# B&R Automation Studio project DosatorePdS
Automation Studio 4.9.6.42 SP; technology packages: mapp 5.24.2, mappView 5.24.0

## Configuration Config1

CPU X20CP1301, AutomationRuntime E4.83, Build 4.1.2, Vc V4.72.6

### Task classes (Cpu.sw)
```
Cyclic#1:
  Program <- Program.prg
Cyclic#4:
  Recipe <- Recipe.prg
Binaries: FWRules, mvLoader, udbdef, TCData, arsvcreg, iomap, sysconf, asfw, User, arconfig, ashwd, Role, ashwac, asnxdb1, Config
Libraries: standard, MpRecipe, MpBase, sys_lib, runtime, MpFile, FileIO, asieccon, astime, arssl, asusb, asbrstr
```

### Hardware
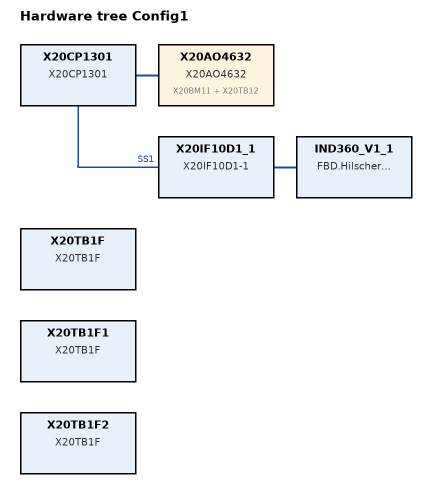
```
IND360_V1_1 : FBD.Hilscher.EIGenEDSAdapterDTM.IND360 V1.1 v1.1 (OrderNumber=IND360 V1.1, VendorAddress=192.168.10.2)  [EIP1 -> X20IF10D1_1.IF1]
  DtmId = a24ae709-e73d-4013-bb43-1e95cdfb2512
  ChannelBlocks_b1ae809b-d69f-462c-9f47-1551c55d3122  // Module 0
  IO_InputImage_b1ae809b-d69f-462c-9f47-1551c55d3122  // 16 Byte(s)
  Channel_1_IO_InputImage_b1ae809b-d69f-462c-9f47-1551c55d3122
  Name_Channel_1_IO_InputImage_b1ae809b-d69f-462c-9f47-1551c55d3122 = MB1_Command_Value
  Type_Channel_1_IO_InputImage_b1ae809b-d69f-462c-9f47-1551c55d3122 = REAL
  Channel_2_IO_InputImage_b1ae809b-d69f-462c-9f47-1551c55d3122
  Name_Channel_2_IO_InputImage_b1ae809b-d69f-462c-9f47-1551c55d3122 = MB1_Channel_Mask
  Type_Channel_2_IO_InputImage_b1ae809b-d69f-462c-9f47-1551c55d3122 = UINT
  Channel_3_IO_InputImage_b1ae809b-d69f-462c-9f47-1551c55d3122
  Name_Channel_3_IO_InputImage_b1ae809b-d69f-462c-9f47-1551c55d3122 = MB1_Command
  Type_Channel_3_IO_InputImage_b1ae809b-d69f-462c-9f47-1551c55d3122 = INT
  Channel_4_IO_InputImage_b1ae809b-d69f-462c-9f47-1551c55d3122
  Name_Channel_4_IO_InputImage_b1ae809b-d69f-462c-9f47-1551c55d3122 = SB1_Reserved_1
  Type_Channel_4_IO_InputImage_b1ae809b-d69f-462c-9f47-1551c55d3122 = INT
  Channel_5_IO_InputImage_b1ae809b-d69f-462c-9f47-1551c55d3122
  Name_Channel_5_IO_InputImage_b1ae809b-d69f-462c-9f47-1551c55d3122 = SB1_Reserved_2
  Type_Channel_5_IO_InputImage_b1ae809b-d69f-462c-9f47-1551c55d3122 = INT
  Channel_6_IO_InputImage_b1ae809b-d69f-462c-9f47-1551c55d3122
  Name_Channel_6_IO_InputImage_b1ae809b-d69f-462c-9f47-1551c55d3122 = SB1_Reserved_3
  Type_Channel_6_IO_InputImage_b1ae809b-d69f-462c-9f47-1551c55d3122 = INT
  Channel_7_IO_InputImage_b1ae809b-d69f-462c-9f47-1551c55d3122
  Name_Channel_7_IO_InputImage_b1ae809b-d69f-462c-9f47-1551c55d3122 = SB1_Command
  Type_Channel_7_IO_InputImage_b1ae809b-d69f-462c-9f47-1551c55d3122 = INT
  IO_OutputImage_b1ae809b-d69f-462c-9f47-1551c55d3122  // 16 Byte(s)
  Channel_1_IO_OutputImage_b1ae809b-d69f-462c-9f47-1551c55d3122
  Name_Channel_1_IO_OutputImage_b1ae809b-d69f-462c-9f47-1551c55d3122 = MB1_Measuring_Value
  Type_Channel_1_IO_OutputImage_b1ae809b-d69f-462c-9f47-1551c55d3122 = REAL
  Channel_2_IO_OutputImage_b1ae809b-d69f-462c-9f47-1551c55d3122
  Name_Channel_2_IO_OutputImage_b1ae809b-d69f-462c-9f47-1551c55d3122 = MB1_Device_Status
  Type_Channel_2_IO_OutputImage_b1ae809b-d69f-462c-9f47-1551c55d3122 = UINT
  Channel_3_IO_OutputImage_b1ae809b-d69f-462c-9f47-1551c55d3122
  Name_Channel_3_IO_OutputImage_b1ae809b-d69f-462c-9f47-1551c55d3122 = MB1_Response
  Type_Channel_3_IO_OutputImage_b1ae809b-d69f-462c-9f47-1551c55d3122 = INT
  Channel_4_IO_OutputImage_b1ae809b-d69f-462c-9f47-1551c55d3122
  Name_Channel_4_IO_OutputImage_b1ae809b-d69f-462c-9f47-1551c55d3122 = SB1_Status_Group_1
  Type_Channel_4_IO_OutputImage_b1ae809b-d69f-462c-9f47-1551c55d3122 = INT
  Channel_5_IO_OutputImage_b1ae809b-d69f-462c-9f47-1551c55d3122
  Name_Channel_5_IO_OutputImage_b1ae809b-d69f-462c-9f47-1551c55d3122 = SB1_Status_Group_2
  Type_Channel_5_IO_OutputImage_b1ae809b-d69f-462c-9f47-1551c55d3122 = INT
  Channel_6_IO_OutputImage_b1ae809b-d69f-462c-9f47-1551c55d3122
  Name_Channel_6_IO_OutputImage_b1ae809b-d69f-462c-9f47-1551c55d3122 = SB1_Status_Group_3
  Type_Channel_6_IO_OutputImage_b1ae809b-d69f-462c-9f47-1551c55d3122 = INT
  Channel_7_IO_OutputImage_b1ae809b-d69f-462c-9f47-1551c55d3122
  Name_Channel_7_IO_OutputImage_b1ae809b-d69f-462c-9f47-1551c55d3122 = SB1_Response
  Type_Channel_7_IO_OutputImage_b1ae809b-d69f-462c-9f47-1551c55d3122 = INT
X20AO4632 : X20AO4632 v1.3.1.0  [SS1 -> X20TB12.SS; SL -> X20BM11.SL1]
  ChannelType01 = 0 to 20mA
X20BM11 : X20BM11 v1.1.0.0  [X2X1 -> X20CP1301.IF6]
X20CP1301 : X20CP1301 v1.7.0.0  [X1 -> X1.SL; X2 -> X2.SL; X3 -> X3.SL]
  Module X1 (Type=X1, Virtual=true, Version=1.7.0.0)
    Connection (Connector=SS1, TargetModule=X20TB1F, TargetConnector=SS)
    Connection (Connector=SL, TargetModule=X20CP1301, TargetConnector=X1)
    X1AI_ChannelType01 = 0 to 20mA
    X1AI1_InputFilter = level 2
    X1AI_ChannelType02 = 0 to 20mA
  Module X2 (Type=X2, Virtual=true, Version=1.7.0.0)
    Connection (Connector=SS1, TargetModule=X20TB1F1, TargetConnector=SS)
    Connection (Connector=SL, TargetModule=X20CP1301, TargetConnector=X2)
  Module X3 (Type=X3, Virtual=true, Version=1.7.0.0)
    Connection (Connector=SS1, TargetModule=X20TB1F2, TargetConnector=SS)
    Connection (Connector=SL, TargetModule=X20CP1301, TargetConnector=X3)
  Connector IF2:
    ActivateDevice = 1
    Mode = Manual
    InternetAddress = 192.168.0.2
    SubnetMask = 255.255.255.0
  ConfigurationID = DosatorePdS_Config1
  UserPartitionSize = 200
  EnableUsbRemoteInstall = 1
  Cyclic1Tolerance = 0
  FileDevice1
  FileDeviceName1 = CF
  FileDevicePath1 = F:\Recipe
  FtpUser1
  FtpUsername1 = bazzica
  FtpUserPassword1 = htUSodyHi80qCEfYHuTU7vQ0j0QXP3jVAlZaBuEyoRs=  // promass
  FtpUserSalt1 = 1uLtMhRf
  FTPAccessRight1 = 0
  ActivateOpcUa = 1
  OpcUaInformationModels_PV_Version = 1
X20IF10D1_1 : X20IF10D1-1 v1.7.0.0  [SS -> X20CP1301.SS1]
  Connector IF1:
    DtmId = ce78e8b2-5855-467c-9c90-e15d78aa6884
  ConfigFile = X20IF10D1_1.dtm
  ConfigModule = asnxdb1
X20TB12 : X20TB12 v1.0.0.0
X20TB1F : X20TB1F v1.0.0.0
X20TB1F1 : X20TB1F v1.0.0.0
X20TB1F2 : X20TB1F v1.0.0.0
```

### IoMap.iom - X20CP1301/IoMap.iom
```iecst
VAR_CONFIG
	Cyclic#1.GlbIO.Ao.Valvola AT %QW."X20AO4632".AnalogOutput01;
	GlbIO.Do.PompaAspirazione AT %QX."X3".DigitalOutput01;
	PesoBilancia_G AT %ID."IND360_V1_1".MB1_Command_Value;
	::GlbIO.Ai.Valvola AT %IW."X1".AnalogInput02;
END_VAR
```

## Configuration Config2

### Task classes (Cpu.sw)
```
Cyclic#1:
  simu <- simu.prg
  Program <- Program.prg
Cyclic#4:
  Recipe <- Recipe.prg
Binaries: FWRules, mvLoader, udbdef, TCData, arsvcreg, iomap, sysconf, asfw, User, arconfig, ashwd, Role, ashwac, asnxdb1, Config
Libraries: standard, MpRecipe, MpBase, sys_lib, runtime, MpFile, FileIO, asieccon, astime, arssl, asusb, asbrstr
```

### Hardware
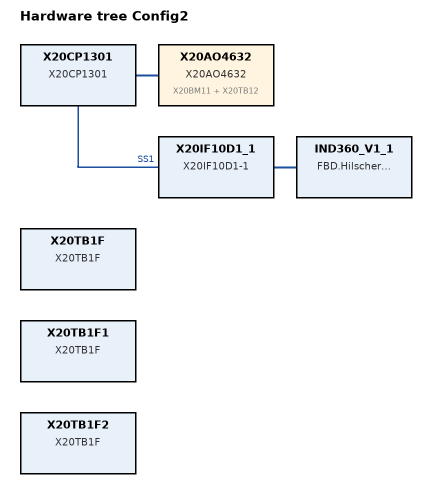
```
IND360_V1_1 : FBD.Hilscher.EIGenEDSAdapterDTM.IND360 V1.1 v1.1 (OrderNumber=IND360 V1.1, VendorAddress=192.168.10.2)  [EIP1 -> X20IF10D1_1.IF1]
  DtmId = a24ae709-e73d-4013-bb43-1e95cdfb2512
  ChannelBlocks_b1ae809b-d69f-462c-9f47-1551c55d3122  // Module 0
  IO_InputImage_b1ae809b-d69f-462c-9f47-1551c55d3122  // 16 Byte(s)
  Channel_1_IO_InputImage_b1ae809b-d69f-462c-9f47-1551c55d3122
  Name_Channel_1_IO_InputImage_b1ae809b-d69f-462c-9f47-1551c55d3122 = MB1_Command_Value
  Type_Channel_1_IO_InputImage_b1ae809b-d69f-462c-9f47-1551c55d3122 = REAL
  Channel_2_IO_InputImage_b1ae809b-d69f-462c-9f47-1551c55d3122
  Name_Channel_2_IO_InputImage_b1ae809b-d69f-462c-9f47-1551c55d3122 = MB1_Channel_Mask
  Type_Channel_2_IO_InputImage_b1ae809b-d69f-462c-9f47-1551c55d3122 = UINT
  Channel_3_IO_InputImage_b1ae809b-d69f-462c-9f47-1551c55d3122
  Name_Channel_3_IO_InputImage_b1ae809b-d69f-462c-9f47-1551c55d3122 = MB1_Command
  Type_Channel_3_IO_InputImage_b1ae809b-d69f-462c-9f47-1551c55d3122 = INT
  Channel_4_IO_InputImage_b1ae809b-d69f-462c-9f47-1551c55d3122
  Name_Channel_4_IO_InputImage_b1ae809b-d69f-462c-9f47-1551c55d3122 = SB1_Reserved_1
  Type_Channel_4_IO_InputImage_b1ae809b-d69f-462c-9f47-1551c55d3122 = INT
  Channel_5_IO_InputImage_b1ae809b-d69f-462c-9f47-1551c55d3122
  Name_Channel_5_IO_InputImage_b1ae809b-d69f-462c-9f47-1551c55d3122 = SB1_Reserved_2
  Type_Channel_5_IO_InputImage_b1ae809b-d69f-462c-9f47-1551c55d3122 = INT
  Channel_6_IO_InputImage_b1ae809b-d69f-462c-9f47-1551c55d3122
  Name_Channel_6_IO_InputImage_b1ae809b-d69f-462c-9f47-1551c55d3122 = SB1_Reserved_3
  Type_Channel_6_IO_InputImage_b1ae809b-d69f-462c-9f47-1551c55d3122 = INT
  Channel_7_IO_InputImage_b1ae809b-d69f-462c-9f47-1551c55d3122
  Name_Channel_7_IO_InputImage_b1ae809b-d69f-462c-9f47-1551c55d3122 = SB1_Command
  Type_Channel_7_IO_InputImage_b1ae809b-d69f-462c-9f47-1551c55d3122 = INT
  IO_OutputImage_b1ae809b-d69f-462c-9f47-1551c55d3122  // 16 Byte(s)
  Channel_1_IO_OutputImage_b1ae809b-d69f-462c-9f47-1551c55d3122
  Name_Channel_1_IO_OutputImage_b1ae809b-d69f-462c-9f47-1551c55d3122 = MB1_Measuring_Value
  Type_Channel_1_IO_OutputImage_b1ae809b-d69f-462c-9f47-1551c55d3122 = REAL
  Channel_2_IO_OutputImage_b1ae809b-d69f-462c-9f47-1551c55d3122
  Name_Channel_2_IO_OutputImage_b1ae809b-d69f-462c-9f47-1551c55d3122 = MB1_Device_Status
  Type_Channel_2_IO_OutputImage_b1ae809b-d69f-462c-9f47-1551c55d3122 = UINT
  Channel_3_IO_OutputImage_b1ae809b-d69f-462c-9f47-1551c55d3122
  Name_Channel_3_IO_OutputImage_b1ae809b-d69f-462c-9f47-1551c55d3122 = MB1_Response
  Type_Channel_3_IO_OutputImage_b1ae809b-d69f-462c-9f47-1551c55d3122 = INT
  Channel_4_IO_OutputImage_b1ae809b-d69f-462c-9f47-1551c55d3122
  Name_Channel_4_IO_OutputImage_b1ae809b-d69f-462c-9f47-1551c55d3122 = SB1_Status_Group_1
  Type_Channel_4_IO_OutputImage_b1ae809b-d69f-462c-9f47-1551c55d3122 = INT
  Channel_5_IO_OutputImage_b1ae809b-d69f-462c-9f47-1551c55d3122
  Name_Channel_5_IO_OutputImage_b1ae809b-d69f-462c-9f47-1551c55d3122 = SB1_Status_Group_2
  Type_Channel_5_IO_OutputImage_b1ae809b-d69f-462c-9f47-1551c55d3122 = INT
  Channel_6_IO_OutputImage_b1ae809b-d69f-462c-9f47-1551c55d3122
  Name_Channel_6_IO_OutputImage_b1ae809b-d69f-462c-9f47-1551c55d3122 = SB1_Status_Group_3
  Type_Channel_6_IO_OutputImage_b1ae809b-d69f-462c-9f47-1551c55d3122 = INT
  Channel_7_IO_OutputImage_b1ae809b-d69f-462c-9f47-1551c55d3122
  Name_Channel_7_IO_OutputImage_b1ae809b-d69f-462c-9f47-1551c55d3122 = SB1_Response
  Type_Channel_7_IO_OutputImage_b1ae809b-d69f-462c-9f47-1551c55d3122 = INT
X20AO4632 : X20AO4632 v1.3.1.0  [SS1 -> X20TB12.SS; SL -> X20BM11.SL1]
  ChannelType01 = 0 to 20mA
X20BM11 : X20BM11 v1.1.0.0  [X2X1 -> X20CP1301.IF6]
X20CP1301 : X20CP1301 v1.7.0.0  [X1 -> X1.SL; X2 -> X2.SL; X3 -> X3.SL]
  Module X1 (Type=X1, Virtual=true, Version=1.7.0.0)
    Connection (Connector=SS1, TargetModule=X20TB1F, TargetConnector=SS)
    Connection (Connector=SL, TargetModule=X20CP1301, TargetConnector=X1)
    X1AI_ChannelType01 = 0 to 20mA
    X1AI1_InputFilter = level 2
    X1AI_ChannelType02 = 0 to 20mA
  Module X2 (Type=X2, Virtual=true, Version=1.7.0.0)
    Connection (Connector=SS1, TargetModule=X20TB1F1, TargetConnector=SS)
    Connection (Connector=SL, TargetModule=X20CP1301, TargetConnector=X2)
  Module X3 (Type=X3, Virtual=true, Version=1.7.0.0)
    Connection (Connector=SS1, TargetModule=X20TB1F2, TargetConnector=SS)
    Connection (Connector=SL, TargetModule=X20CP1301, TargetConnector=X3)
  Connector IF2:
    ActivateDevice = 1
    Mode = Manual
    InternetAddress = 192.168.0.2
    SubnetMask = 255.255.255.0
  ConfigurationID = DosatorePdS_Config1
  UserPartitionSize = 200
  Simulation = 1
  EnableUsbRemoteInstall = 1
  Cyclic1Tolerance = 0
  FileDevice1
  FileDeviceName1 = CF
  FileDevicePath1 = F:\Recipe
  FtpUser1
  FtpUsername1 = bazzica
  FtpUserPassword1 = htUSodyHi80qCEfYHuTU7vQ0j0QXP3jVAlZaBuEyoRs=  // promass
  FtpUserSalt1 = 1uLtMhRf
  FTPAccessRight1 = 0
  ActivateOpcUa = 1
  OpcUaInformationModels_PV_Version = 1
X20IF10D1_1 : X20IF10D1-1 v1.7.0.0  [SS -> X20CP1301.SS1]
  Connector IF1:
    DtmId = ce78e8b2-5855-467c-9c90-e15d78aa6884
  ConfigFile = X20IF10D1_1.dtm
  ConfigModule = asnxdb1
X20TB12 : X20TB12 v1.0.0.0
X20TB1F : X20TB1F v1.0.0.0
X20TB1F1 : X20TB1F v1.0.0.0
X20TB1F2 : X20TB1F v1.0.0.0
```

### IoMap.iom - X20CP1301/IoMap.iom
```iecst
VAR_CONFIG
	Cyclic#1.GlbIO.Ao.Valvola AT %QW."X20AO4632".AnalogOutput01;
	GlbIO.Do.PompaAspirazione AT %QX."X3".DigitalOutput01;
END_VAR
```

## Logical view

Binary libraries used (declarations not repeated): operator, runtime, astime, AsIecCon, standard, MpRecipe 5.24.2, MpBase 5.24.1, sys_lib, MpFile 5.24.2, FileIO

### Global.typ - Global data types
```iecst
TYPE
	TypDo : 	STRUCT
		PompaAspirazione : BOOL;
	END_STRUCT;
	TypAi : 	STRUCT
		Valvola : INT;
		Bilancia : INT;
	END_STRUCT;
	TypAo : 	STRUCT
		Valvola : INT;
	END_STRUCT;
	TypIO : 	STRUCT
		Ai : TypAi;
		Ao : TypAo;
		Do : TypDo;
	END_STRUCT;
	Typ_recipe : 	STRUCT
		PesoRichiesto : REAL;
		fPesoAnticipoChiusura : REAL;
		fSogliaDosaggioLento : REAL;
		fSogliaMicrodosaggio : REAL;
		fPercentualeValvolaVeloce : REAL;
		fPercentualeValvolaLenta : REAL;
		fPercentualeValvolaFine : REAL;
		fFattoreCorrezione : REAL;
	END_STRUCT;
END_TYPE
```

### Global.var - Global variables
```iecst
VAR
	GlbIO : TypIO;
	Recipe : Typ_recipe;
	PesoBilancia_G : REAL; (*// Peso finale in grammi*)
END_VAR
```


### Program Logical/Program (IEC)

#### Cyclic.st - Cyclic code
```iecst
PROGRAM _CYCLIC
// #######################################################################
// --- LOGICA PRINCIPALE E CALIBRAZIONE ---
// #######################################################################

	IF PercentualeValvola > 0 THEN
		radialGauge := REAL_TO_INT(PercentualeValvola*10);
	ELSE
		radialGauge := 0;
	END_IF

	// conversione segnale d'ingresso valvola

	PercentualeValvola := (((INT_TO_REAL(GlbIO.Ai.Valvola) - 6553.0) / (32767.0 - 6553.0)) * 100.0);

// --- ESECUZIONE TIMER ---
	TON_AttesaStabilizzazione(IN := bStartTimerCal, PT := REAL_TO_TIME(fDurataTestSec * 1000.0));
	TON_AttesaStabilizzazione;

	// --- MAPPATURA I/O e CHIAMATA AL BLOCCO FUNZIONE ---
	PesoBilancia_AI := GlbIO.Ai.Bilancia;
	GlbIO.Ao.Valvola := REAL_TO_INT(Valvola_AO);

	IF Pulsante_Tara THEN Pulsante_Tara := FALSE; PesoTara := PesoBilancia_G; END_IF
	PesoBilancia_G := PesoBilancia_G - PesoTara;

	IF Stop_HMI THEN Dosatore.bFermaDosaggo := 1; ELSE Dosatore.bFermaDosaggo := 0; END_IF
	TON_timerDosaggio;
	TON_timerDosaggio.PT := T#500s;

	IF NOT (Dosatore.eStatoDosaggio = eST_ERRORE OR Dosatore.eStatoDosaggio = eST_COMPLETATO OR Dosatore.eStatoDosaggio = eST_IDLE) THEN
		TON_timerDosaggio.IN := TRUE;
		tDosaggio_HMI := TIME_TO_REAL(TON_timerDosaggio.ET) / 1000;
	ELSE
		TON_timerDosaggio.IN := FALSE;
	END_IF

	Dosatore.fPesoAnticipoChiusura 			:= Recipe.fPesoAnticipoChiusura;
	Dosatore.fSogliaDosaggioLento 			:= Recipe.fSogliaDosaggioLento;
	Dosatore.fSogliaMicrodosaggio 			:= Recipe.fSogliaMicrodosaggio;
	Dosatore.fPercentualeValvolaVeloce 		:= Recipe.fPercentualeValvolaVeloce;
	Dosatore.fPercentualeValvolaLenta 		:= Recipe.fPercentualeValvolaLenta;
	Dosatore.fPercentualeValvolaFine 		:= Recipe.fPercentualeValvolaFine;
	Dosatore.fFattoreCorrezione 			:= Recipe.fFattoreCorrezione;
	Dosatore.fFeadbackValvolaProporzionale 	:= PercentualeValvola;
	PesoRichiesto_HMI						:= Recipe.PesoRichiesto;

	Dosatore(
		fPesoAttualeBilancia := PesoBilancia_G,
		fPesoRichiesto := PesoRichiesto_HMI,
		bAvviaDosaggio := StartDosaggio_HMI
		);

	Recipe.fPesoAnticipoChiusura := Dosatore.fPesoAnticipoChiusura;

	BilanciaManager(
		iRawInput := PesoBilancia_AI,
		bComandoTare := Pulsante_Tara
		// fCapacitaMaxG e iRawMax usano i valori di default (5000.0, 32767) se non specificati
		);

	// Mappa l'uscita
	// PesoBilancia_G := BilanciaManager.fPesoGrammi;

	Valvola_AO := (Dosatore.fUscitaValvolaProporzionale * (32767 - 6600) / 100) + 6600;

	// --- SEQUENZA DI MISURAZIONE DELLA PORTATA ---
	// Logica per eseguire il test di portata con Timer e chiusura valvola
	IF eStatoCalibrazione = eCAL_TEST_PUNTO1_BASSO OR eStatoCalibrazione = eCAL_TEST_PUNTO2_ALTO THEN
	(*	bStartTimerCal := FALSE;*)
		IF NOT TON_AttesaStabilizzazione.Q THEN
			// La variabile Veloce qui funge da variabile temporanea per l'apertura in test
			GlbIO.Ao.Valvola := REAL_TO_INT(Dosatore.fPercentualeValvolaVeloce * 32767 / 100);
		ELSE
			GlbIO.Ao.Valvola := REAL_TO_INT(10000.0);
		END_IF

		// Calcolo della portata dopo il timeout + 10s di stabilizzazione
		IF TON_AttesaStabilizzazione.Q AND TON_AttesaStabilizzazione.ET >= REAL_TO_TIME((fDurataTestSec) * 1000.0) THEN
			fPortataMisurata := (PesoBilancia_G - fPesoIniziale) / fDurataTestSec;
			bStartTimerCal := FALSE; // Termina il test
		END_IF
	END_IF

	// #######################################################################
	// --- MACCHINA A STATI DI CALIBRAZIONE ---
	// #######################################################################

	IF bStartCalibrazione AND NOT bCalibrazioneCompletata THEN

		CASE eStatoCalibrazione OF

			eCAL_IDLE:
				bStartTimerCal := FALSE;
				//Bilancia.Tare := TRUE;
				Dosatore.fFattoreCorrezione := 0.0; // Disabilita l'auto-tuning
				eStatoCalibrazione := eCAL_PREPARA_TEST;

			eCAL_PREPARA_TEST:
				fPortataMisurata := 0.0;
				fPesoIniziale := 0.0;
				eStatoCalibrazione := eCAL_TEST_PUNTO1_BASSO;

				fPesoIniziale := PesoBilancia_G;
				bStartTimerCal := TRUE;

			eCAL_TEST_PUNTO1_BASSO:
				// TEST 1: Misura della portata al punto P1 (20% apertura)
				Dosatore.fPercentualeValvolaVeloce := fPercentualeTestBasso;

//					fPesoIniziale := PesoBilancia_G;
//					bStartTimerCal := TRUE;
				IF NOT bStartTimerCal AND (fPortataMisurata > 0.0) THEN
					fPortataTestBasso := fPortataMisurata;
					eStatoCalibrazione := eCAL_TEST_PUNTO2_ALTO;

					fPesoIniziale := PesoBilancia_G;
					fPortataMisurata := 0;
					bStartTimerCal := TRUE;
				END_IF

			eCAL_TEST_PUNTO2_ALTO:
				// TEST 2: Misura della portata al punto P2 (80% apertura)
				Dosatore.fPercentualeValvolaVeloce := fPercentualeTestAlto;

//					fPesoIniziale := PesoBilancia_G;
//					bStartTimerCal := TRUE;
				IF NOT bStartTimerCal AND (fPortataMisurata > 0.0) THEN
					fPortataTestAlto := fPortataMisurata;
					eStatoCalibrazione := eCAL_CALCOLA_CURVA;
				END_IF

			eCAL_CALCOLA_CURVA:
				// Calcolo dei coefficienti della curva lineare (Percentuale = m * Portata + q)
				IF (fPortataTestAlto - fPortataTestBasso) > 0.001 THEN
					fPendenza_m := (fPercentualeTestAlto - fPercentualeTestBasso) /
					(fPortataTestAlto - fPortataTestBasso);
					fIntercetta_q := fPercentualeTestBasso - (fPendenza_m * fPortataTestBasso);

					eStatoCalibrazione := eCAL_MISURA_VOLO;
				ELSE
					eStatoCalibrazione := eCAL_ERRORE; // Errore: Le portate sono uguali o zero
				END_IF

			eCAL_MISURA_VOLO:
				// CRUCIALE: Misura il peso in volo (forza Dosatore.fPesoAnticipoChiusura = 0.0)
				Dosatore.fPesoAnticipoChiusura := 0.0;
				fSetPointTaratura := 2000.0;
				PesoRichiesto_HMI := fSetPointTaratura;

				StartDosaggio_HMI := TRUE;

				IF Dosatore.bDosaggioCompletato THEN
					StartDosaggio_HMI := FALSE;
					bStartTimerCal := TRUE;
					eStatoCalibrazione := eCAL_ATTESA_PESO;
				END_IF

			eCAL_ATTESA_PESO:
				// Attende stabilizzazione e calcola il volo
				IF TON_AttesaStabilizzazione.Q THEN
					bStartTimerCal := FALSE;

					fAnticipoMisurato := PesoBilancia_G - fSetPointTaratura;

					IF fAnticipoMisurato < 0.5 THEN fAnticipoMisurato := 0.5; END_IF

					eStatoCalibrazione := eCAL_APPLICA_VALORI;
				END_IF

			eCAL_APPLICA_VALORI:
				// Applica i valori tarati al blocco funzione
				Dosatore.fPesoAnticipoChiusura := fAnticipoMisurato;

				// Applica le percentuali dalla curva di calibrazione:
				Dosatore.fPercentualeValvolaVeloce := (fPendenza_m * fPortataTargetVeloce) + fIntercetta_q;
				Dosatore.fPercentualeValvolaLenta := (fPendenza_m * fPortataTargetLenta) + fIntercetta_q;
				Dosatore.fPercentualeValvolaFine := (fPendenza_m * fPortataTargetFine) + fIntercetta_q;

				// Limitazioni di sicurezza
				IF Dosatore.fPercentualeValvolaVeloce > 100.0 THEN Dosatore.fPercentualeValvolaVeloce := 100.0; END_IF
				IF Dosatore.fPercentualeValvolaFine < 0.0 THEN Dosatore.fPercentualeValvolaFine := 0.0; END_IF

				// Ripristina l'auto-taratura continua
				Dosatore.fFattoreCorrezione := 0.1;

				eStatoCalibrazione := eCAL_COMPLETATO;

			eCAL_COMPLETATO:
				bCalibrazioneCompletata := TRUE;
				eStatoCalibrazione := eCAL_IDLE;

			eCAL_ERRORE:
			// ... Logica di errore

		END_CASE

	END_IF

	IF GlbIO.Ao.Valvola < 6500 THEN GlbIO.Ao.Valvola := 6500; END_IF

END_PROGRAM
```

#### Init.st - Init code
```iecst
PROGRAM _INIT
	(* Insert code here *)

	IF bCalibrazioneCompletata THEN
		// Applica i valori tarati al blocco funzione
		Dosatore.fPesoAnticipoChiusura := fAnticipoMisurato;

		// Applica le percentuali dalla curva di calibrazione:
		Dosatore.fPercentualeValvolaVeloce := (fPendenza_m * fPortataTargetVeloce) + fIntercetta_q;
		Dosatore.fPercentualeValvolaLenta := (fPendenza_m * fPortataTargetLenta) + fIntercetta_q;
		Dosatore.fPercentualeValvolaFine := (fPendenza_m * fPortataTargetFine) + fIntercetta_q;

		// Limitazioni di sicurezza
		IF Dosatore.fPercentualeValvolaVeloce > 100.0 THEN Dosatore.fPercentualeValvolaVeloce := 100.0; END_IF
		IF Dosatore.fPercentualeValvolaFine < 0.0 THEN Dosatore.fPercentualeValvolaFine := 0.0; END_IF

		// Ripristina l'auto-taratura continua
		Dosatore.fFattoreCorrezione := 0.1;
	END_IF

END_PROGRAM
```

#### Types.typ - Local data types
```iecst
TYPE
	enSignalType :
		(
		eST_0_20mA,
		eST_4_20mA
		);
	enStatoDosaggio :
		(
		eST_IDLE := 10,
		eST_VELOCE := 20,
		eST_LENTO := 30,
		eST_FINE := 40,
		eST_ATTESA_STABILIZZAZIONE := 50,
		eST_COMPLETATO := 60,
		eST_ERRORE := 0
		);
	enStatoCalibrazione :
		( (*// Macchina a Stati per la Calibrazione*)
		eCAL_IDLE := 10,
		eCAL_PREPARA_TEST := 20,
		eCAL_TEST_PUNTO1_BASSO,
		eCAL_TEST_PUNTO2_ALTO,
		eCAL_CALCOLA_CURVA,
		eCAL_MISURA_VOLO := 30,
		eCAL_ATTESA_PESO := 40,
		eCAL_APPLICA_VALORI := 50,
		eCAL_COMPLETATO := 60,
		eCAL_ERRORE := 0
		);
END_TYPE
```

#### Variables.var - Local variables
```iecst
VAR
	tDosaggio_HMI : REAL;
	TON_timerDosaggio : TON;
	PercentualeValvola : REAL;
END_VAR
VAR RETAIN
	Dosatore : FB_DosaggioPolvere; (*// Istanza del blocco funzione*)
END_VAR
VAR
	PesoBilancia_AI : INT; (*// Ingresso Analogico (da I/O Link o bus)*)
	Valvola_AO : REAL; (*// Uscita Analogica (verso I/O Link o bus)*)
	Stop_HMI : BOOL;
END_VAR
VAR RETAIN
	PesoRichiesto_HMI : REAL; (*// Setpoint (da HMI)*)
END_VAR
VAR
	StartDosaggio_HMI : BOOL; (*// Tasto Start (da HMI)*)
	DosaggioOK : BOOL; (*// Stato di completamento*) (*// --- VARIABILI PER LA TARATURA AUTOMATICA ---*)
	bStartCalibrazione : BOOL; (*// Comando esterno per avviare la taratura (es. da HMI)*)
END_VAR
VAR RETAIN
	bCalibrazioneCompletata : BOOL;
END_VAR
VAR
	eStatoCalibrazione : enStatoCalibrazione; (*// Macchina a Stati per la Calibrazione*) (*// Variabili interne per la Taratura*)
END_VAR
(*// Parametri della Curva e Portate Target*)
VAR
	fPortataTestBasso : REAL;
	fPortataTestAlto : REAL;
	fPercentualeTestBasso : REAL := 45;
	fPercentualeTestAlto : REAL := 80.0;
END_VAR
VAR RETAIN
	fPendenza_m : REAL;
	fIntercetta_q : REAL;
END_VAR
VAR
	fPortataTargetVeloce : REAL := 80.0; (*// Target di flusso in g/s per Veloce*)
	fPortataTargetLenta : REAL := 15.0; (*// Target di flusso in g/s per Lenta*)
	fPortataTargetFine : REAL := 5.0; (*// Target di flusso in g/s per Fine*)
END_VAR
(*// Variabili interne*)
VAR
	fAnticipoMisurato : REAL; (*// Risultato del test di misurazione del volo*)
	fSetPointTaratura : REAL; (*// Setpoint specifico per il test*)
	fPortataMisurata : REAL; (*// Portata misurata in [grammi/secondo]*)
	fPesoIniziale : REAL;
	fDurataTestSec : REAL := 5; (*// Durata di ogni test di portata (3 secondi)*)
END_VAR
(*// Timer e Logica Timer*)
VAR
	TON_AttesaStabilizzazione : TON; (*// Timer per attendere che la bilancia si stabilizzi*)
	bStartTimerCal : BOOL := FALSE;
	ModuloBilancia_Raw : INT; (*// Dati grezzi in ingresso (dall'I/O)*)
END_VAR
VAR RETAIN
	PesoTara : REAL;
END_VAR
VAR
	Pulsante_Tara : BOOL; (*// Comando di azzeramento da HMI o logica*)
END_VAR
VAR RETAIN
	BilanciaManager : FB_GestioneBilancia; (*// Istanza del Blocco Funzione*)
END_VAR
VAR
	radialGauge : UINT;
END_VAR
```

#### LocalFunctions.fun
```iecst
FUNCTION_BLOCK FB_GestioneBilancia
	VAR_INPUT
		iRawInput : INT; (*// Ingresso: Valore raw (grezzo) letto dal modulo I/O (es. 0 a 32767)*)
		bComandoTare : BOOL; (*// Ingresso: Commuta a TRUE per eseguire l'azzeramento (Tara)*)
		eTipoSegnale : enSignalType := eST_4_20mA; (*/ NUOVO: Tipo di segnale (0-20mA o 4-20mA)*)
		fCapacitaMaxG : REAL := 6000.0; (*// Ingresso: Capacità massima della bilancia in grammi*)
		iRawMax : INT := 32767; (*// Ingresso: Valore massimo raw del modulo I/O*)
	END_VAR
	VAR_OUTPUT
		bErroreSegnale : BOOL;
		fPesoGrammi : REAL; (*// Uscita: Peso convertito e tarato in grammi (REAL)*)
	END_VAR
	VAR
		fFattoreConversione : REAL; (*// Fattore per convertire Raw in Grammi/Volt*)
		fOffsetTara : REAL := 0.0; (*// Offset di tara (peso memorizzato durante l'azzeramento)*)
		fPesoLordoSenzaOffset : REAL; (*// Peso convertito prima dell'applicazione della tara*)
		iRawMin : INT; (*// Valore raw minimo corrispondente a 0mA o 4mA*)
		iRawRange : INT; (*// RawMax - RawMin*)
		fRawAttualeNormalizzato : REAL; (*// Raw letto - RawMin*)
	END_VAR
END_FUNCTION_BLOCK

{REDUND_ERROR} FUNCTION_BLOCK FB_DosaggioPolvere
	VAR_INPUT
		fPesoAttualeBilancia : REAL; (*// Ingresso: Peso letto dalla bilancia (es. in grammi)*)
		fPesoRichiesto : REAL; (*// Ingresso: Setpoint del peso desiderato (es. in grammi)*)
		bFermaDosaggo : BOOL; (*// Ingresso: Commuta a TRUE per iniziare il ciclo*) (*// --- PARAMETRI DI PRECISIONE ---*)
		bAvviaDosaggio : BOOL; (*// Ingresso: Commuta a TRUE per iniziare il ciclo*) (*// --- PARAMETRI DI PRECISIONE ---*)
		fTolleranzaPercentuale : REAL := 0.0005; (*Fattore per lo 0.05% (0.05 / 100)*)
		fPesoAnticipoChiusura : REAL := 5.0; (*Ingresso: Peso (in grammi) che è in volo dopo la chiusura della valvola (DEVE ESSERE CALIBRATO!)*) (*// --- PARAMETRI DI FASE ---*)
		fSogliaDosaggioLento : REAL := 0.90; (*// Ingresso: Percentuale del setpoint per passare a dosaggio lento (es. 90%)*)
		fSogliaMicrodosaggio : REAL := 0.97; (*// Ingresso: Percentuale del setpoint per passare a microdosaggio (es. 99%)*)
		fPercentualeValvolaVeloce : REAL := 70.0; (*// Ingresso: Apertura valvola per dosaggio veloce (0-100)*)
		fPercentualeValvolaLenta : REAL := 50; (*// Ingresso: Apertura valvola per dosaggio lento (0-100)*)
		fPercentualeValvolaFine : REAL := 47; (*// Ingresso: Apertura valvola per microdosaggio (0-100)*)
		tTimeoutStabilizzazione : TIME := T#5s; (*Tempo massimo di attesa per la stabilizzazione (es. 5 secondi)*)
		fFattoreCorrezione : REAL := 0.1; (*Fattore che determina la velocità di correzione (es. 0.1 = correggiamo il 10% dell'errore ad ogni ciclo)*)
		C_CAPACITA_MAX_BILANCIA : REAL := 3500;
		fFeadbackValvolaProporzionale : REAL; (*// Uscita: Comando alla valvola proporzionale (0.0 - 100.0)*)
	END_VAR
	VAR_OUTPUT
		fUscitaValvolaProporzionale : REAL; (*// Uscita: Comando alla valvola proporzionale (0.0 - 100.0)*)
		bDosaggioCompletato : BOOL; (*// Uscita: TRUE quando il dosaggio è finito e preciso*)
		bDosaggioInCorso : BOOL; (*// Uscita: TRUE durante il ciclo di dosaggio*)
		bErroreStabilizzazione : BOOL; (*TRUE se il dosaggio è fallito per timeout*)
		eStatoDosaggio : enStatoDosaggio; (*// Stato macchina*)
	END_VAR
	VAR
		fPesoTargetVeloce : REAL; (*// Peso limite per dosaggio veloce*)
		fPesoTargetLento : REAL; (*// Peso limite per dosaggio lento*)
		fErrorePercentuale : REAL; (*// Errore calcolato in %*)
		fSetPointErrore : REAL;
		fTolleranzaMinima : REAL; (*Limite inferiore accettabile*)
		fTolleranzaMassima : REAL; (*Limite superiore accettabile*)
		fPuntoDiChiusuraValvola : REAL; (*Nuovo punto di chiusura calcolato*) (*// VARIABILI TIMER*)
		bStartTimerAttesa : BOOL; (*Flag per attivare il timer*)
		bStartTimer : BOOL; (*Flag per attivare il timer*)
		TON_AttesaMateriale : TON; (*Istanza del Timer di Attesa, dopo questo tempo, se il materiale non passaaumento l'apertura della valvola*) (*// VARIABILI PER L'AUTO-TARATURA*)
		TON_Stabilizzazione : TON; (*Istanza del Timer On Delay*) (*// VARIABILI PER L'AUTO-TARATURA*)
		fUltimoPesoDosato : REAL; (*Peso finale registrato nel ciclo precedente*)
		fUltimoErroreAssoluto : REAL; (*Differenza tra fUltimoPesoDosato e fPesoRichiesto*)
		fErroreAssolutoMax : REAL; (*// Valore calcolato: Peso max di errore (es. 1.0g per 2000g)*)
		fOldWeight : REAL; (*vecchio valore bilancia per controllo flusso*)
		fIncrementoPercentualeValvola : REAL;
		fPercentualeValvolaPrec : REAL;
		fPortataAlComandoChiusura : REAL;
		fPortataAttuale : REAL;
		fFattoreCorrezioneValvola : REAL;
		fMaterialeInVolo : REAL;
		fTempoRitardoStimato : REAL;
		fPesoAlComandoChiusura : REAL;
		fMaterialeCadutoDopoChiusura : REAL;
		fTempoRitardoPrecedente : REAL;
		bilanciaPortataOld : REAL;
	END_VAR
END_FUNCTION_BLOCK
```

#### FB_DosaggioPolvere.st
```iecst
FUNCTION_BLOCK FB_DosaggioPolvere

	// --- CONTROLLO GUASTI DI SICUREZZA ---
	IF fPesoAttualeBilancia < -10.0 OR fPesoAttualeBilancia > C_CAPACITA_MAX_BILANCIA THEN
		eStatoDosaggio := eST_ERRORE;
	END_IF

	IF bFermaDosaggo THEN eStatoDosaggio := eST_IDLE; END_IF;

	// --- ESECUZIONE TIMER E CALCOLI PRELIMINARI ---
	TON_Stabilizzazione(IN := bStartTimer, PT := tTimeoutStabilizzazione);
	TON_AttesaMateriale(IN := bStartTimerAttesa, PT := T#2s);

	// CALCOLO DELL'ERRORE MASSIMO ASSOLUTO (basato sulla percentuale)
	fErroreAssolutoMax := fPesoRichiesto * fTolleranzaPercentuale;

	// Calcolo del Punto di Chiusura (Anticipo del Volo)
	//fPuntoDiChiusuraValvola := fPesoRichiesto - fPesoAnticipoChiusura;
	fTempoRitardoPrecedente := fPesoAnticipoChiusura;

	// Calcolo dei Target
	fPesoTargetVeloce := (fPesoRichiesto) * fSogliaDosaggioLento/100;
	fPesoTargetLento := (fPesoRichiesto) * fSogliaMicrodosaggio/100;

	// Calcolo dei Limiti di Tolleranza Finale
	fTolleranzaMinima := fPesoRichiesto - fErroreAssolutoMax;
	fTolleranzaMassima := fPesoRichiesto + fErroreAssolutoMax;

	fPortataAttuale := (fPesoAttualeBilancia - bilanciaPortataOld)/0.01;
	bilanciaPortataOld := fPesoAttualeBilancia;

	IF NOT TON_AttesaMateriale.Q THEN
		fOldWeight := fPesoAttualeBilancia;
	END_IF

	// Gestione degli stati
	CASE eStatoDosaggio OF

		eST_IDLE: // Stato di riposo, attende il comando di avvio
			bStartTimer := FALSE; // Timer disattivo
			bErroreStabilizzazione := FALSE;
			bDosaggioInCorso := FALSE;
			bDosaggioCompletato := FALSE;
			fUscitaValvolaProporzionale := 0.0; // Valvola chiusa
			fIncrementoPercentualeValvola:= 0;

			IF bAvviaDosaggio AND (fPesoRichiesto > 0.0) THEN
				eStatoDosaggio := eST_VELOCE;
				bDosaggioInCorso := TRUE;
			END_IF

		eST_VELOCE: // Dosaggio Veloce (fino al 90% del peso richiesto)
			bStartTimer := FALSE; // Timer disattivo
			fUscitaValvolaProporzionale := fPercentualeValvolaVeloce + fIncrementoPercentualeValvola; // Apertura valvola al valore veloce

			IF fUscitaValvolaProporzionale > 100 THEN
				eStatoDosaggio := eST_ERRORE;
			END_IF

			IF ABS(fUscitaValvolaProporzionale - fFeadbackValvolaProporzionale) < 5 THEN
				bStartTimerAttesa := TRUE;
				IF TON_AttesaMateriale.Q AND (ABS(fOldWeight - fPesoAttualeBilancia) < 5) THEN
					fIncrementoPercentualeValvola := fIncrementoPercentualeValvola + 7;
				END_IF
			ELSE
				bStartTimerAttesa := FALSE;
			END_IF

			// Transizione allo stato successivo
			IF fPesoAttualeBilancia >= fPesoTargetVeloce THEN
				eStatoDosaggio := eST_LENTO;
				fIncrementoPercentualeValvola:= 0;
			END_IF

		eST_LENTO: // Dosaggio Lento (dal 90% al 99% del peso richiesto)
			bStartTimer := FALSE; // Timer disattivo
			fUscitaValvolaProporzionale := fPercentualeValvolaLenta + fIncrementoPercentualeValvola; // Apertura valvola al valore lento per maggiore precisione

			IF fUscitaValvolaProporzionale > 100 THEN
				eStatoDosaggio := eST_ERRORE;
			END_IF

			IF ABS(fUscitaValvolaProporzionale - fFeadbackValvolaProporzionale) < 4 THEN
				bStartTimerAttesa := TRUE;
				IF TON_AttesaMateriale.Q AND (ABS(fOldWeight - fPesoAttualeBilancia) < 4) THEN
					fIncrementoPercentualeValvola := fIncrementoPercentualeValvola + 5;
				END_IF
			ELSE
				bStartTimerAttesa := FALSE;
			END_IF

			// Transizione allo stato successivo
			IF fPesoAttualeBilancia >= fPesoTargetLento THEN
				eStatoDosaggio := eST_FINE;
				fIncrementoPercentualeValvola:= 0;
			END_IF

		eST_FINE: // Microdosaggio (dal 99% fino al punto di chiusura anticipata)

			// --- 1. CALCOLO DINAMICO DEL PUNTO DI CHIUSURA ---
			IF fPercentualeValvolaPrec > 0.0 THEN
				fFattoreCorrezioneValvola := fFeadbackValvolaProporzionale / fPercentualeValvolaPrec;
			ELSE
				fFattoreCorrezioneValvola := 1.0; // Sicurezza per il primo ciclo assoluto
			END_IF

			// Stima del ritardo e del materiale in volo (Anticipo dinamico)
			fTempoRitardoStimato := fTempoRitardoPrecedente * fFattoreCorrezioneValvola;
			fMaterialeInVolo := fPortataAttuale * fTempoRitardoStimato;
			fPuntoDiChiusuraValvola := fPesoRichiesto - fMaterialeInVolo;
			// --------------------------------------------------

			fUscitaValvolaProporzionale := fPercentualeValvolaFine + fIncrementoPercentualeValvola; // Apertura minima della valvola (Microdosaggio)

			IF fUscitaValvolaProporzionale > 100 THEN
				eStatoDosaggio := eST_ERRORE;
			END_IF

			IF fPortataAttuale < 2 THEN
				bStartTimerAttesa := TRUE;
				IF TON_AttesaMateriale.Q AND (ABS(fOldWeight - fPesoAttualeBilancia) < 2) THEN
					fIncrementoPercentualeValvola := fIncrementoPercentualeValvola + 3;
				END_IF
			ELSE
				bStartTimerAttesa := FALSE;
			END_IF

			// --- 2. CONDIZIONE DI CHIUSURA ANTICIPATA ---
			IF fPesoAttualeBilancia >= fPuntoDiChiusuraValvola THEN

				// SALVATAGGIO DATI PER L'AUTO-APPRENDIMENTO DEL CICLO SUCCESSIVO
				fPercentualeValvolaPrec := fFeadbackValvolaProporzionale;
				fPortataAlComandoChiusura := fPortataAttuale;
				fPesoAlComandoChiusura := fPesoAttualeBilancia;

				fUscitaValvolaProporzionale := 0.0;	// Chiusura IMMEDIATA della valvola
				bStartTimer := TRUE; // AVVIO DEL TIMER e transizione allo stato di attesa
				eStatoDosaggio := eST_ATTESA_STABILIZZAZIONE; // Passaggio ad uno stato di attesa per la stabilizzazione/volo
				fIncrementoPercentualeValvola:= 0;
			END_IF

		eST_ATTESA_STABILIZZAZIONE: // Stato di attesa: la valvola è chiusa (Output = 0.0), il timer è attivo
			bStartTimer := TRUE; // Mantiene attivo l'ingresso del TON

			// Controllo di successo: Peso stabilizzato nell'intervallo ACCETTABILE
			IF fPesoAttualeBilancia >= fTolleranzaMinima AND fPesoAttualeBilancia <= fTolleranzaMassima AND TON_Stabilizzazione.Q THEN
				bStartTimer := FALSE;
				eStatoDosaggio := eST_COMPLETATO;

				// --- LOGICA DI AUTO-TARATURA (SUCCESSO) ---
				IF fPortataAlComandoChiusura > 0.0 THEN
					fMaterialeCadutoDopoChiusura := fPesoAttualeBilancia - fPesoAlComandoChiusura;
					fTempoRitardoPrecedente := fMaterialeCadutoDopoChiusura / fPortataAlComandoChiusura;
				END_IF

			ELSIF TON_Stabilizzazione.Q THEN
				// Controllo di errore: Timeout raggiunto e peso fuori tolleranza

				bStartTimer := FALSE; // Spegne il timer
				bErroreStabilizzazione := TRUE; // Segnala l'errore specifico
				//eStatoDosaggio := eST_ERRORE;

				// --- LOGICA DI AUTO-TARATURA (ERRORE) ---
				// Anche se è in errore, calcoliamo il ritardo reale per correggere il prossimo ciclo
				IF fPortataAlComandoChiusura > 0.0 THEN
					fMaterialeCadutoDopoChiusura := fPesoAttualeBilancia - fPesoAlComandoChiusura;

					// Protezione per evitare calcoli errati se qualcuno ha toccato la bilancia
					IF fMaterialeCadutoDopoChiusura > 0.0 THEN
						fTempoRitardoPrecedente := fMaterialeCadutoDopoChiusura / fPortataAlComandoChiusura;
						eStatoDosaggio := eST_ERRORE;
					END_IF
				END_IF

				// Registra l'ultimo risultato per diagnostica o per HMI
				fUltimoPesoDosato := fPesoAttualeBilancia;
				fUltimoErroreAssoluto := fUltimoPesoDosato - fPesoRichiesto;
			END_IF

			//		eST_FINE: // Microdosaggio (dal 99% fino al punto di chiusura anticipata)
			//			fUscitaValvolaProporzionale := fPercentualeValvolaFine + fIncrementoPercentualeValvola; // Apertura minima della valvola (Microdosaggio)
			//
			//			IF fUscitaValvolaProporzionale > 100 THEN
			//				eStatoDosaggio := eST_ERRORE;
			//			END_IF
			//
			//			IF ABS(fUscitaValvolaProporzionale - fFeadbackValvolaProporzionale) < 2 THEN
			//				bStartTimerAttesa := TRUE;
			//				IF TON_AttesaMateriale.Q AND (ABS(fOldWeight - fPesoAttualeBilancia) < 2) THEN
			//					fIncrementoPercentualeValvola := fIncrementoPercentualeValvola + 3;
			//				END_IF
			//			ELSE
			//				bStartTimerAttesa := FALSE;
			//			END_IF
			//
			//			// CONDIZIONE DI CHIUSURA ANTICIPATA:
			//			IF fPesoAttualeBilancia >= fPuntoDiChiusuraValvola THEN
			//
			//				fUscitaValvolaProporzionale := 0.0;	// Chiusura IMMEDIATA della valvola
			//				bStartTimer := TRUE; // AVVIO DEL TIMER e transizione allo stato di attesa
			//				eStatoDosaggio := eST_ATTESA_STABILIZZAZIONE; // Passaggio ad uno stato di attesa per la stabilizzazione/volo
			//				fIncrementoPercentualeValvola:= 0;
			//			END_IF
			//
			//		eST_ATTESA_STABILIZZAZIONE: // Stato di attesa: la valvola è chiusa (Output = 0.0), il timer è attivo
			//			bStartTimer := TRUE; // Mantiene attivo l'ingresso del TON
			//
			//			// 1. Controllo di successo: Peso stabilizzato nell'intervallo ACCETTABILE (0.05% del setpoint)
			//			IF fPesoAttualeBilancia >= fTolleranzaMinima AND fPesoAttualeBilancia <= fTolleranzaMassima AND TON_Stabilizzazione.Q THEN
			//				bStartTimer := FALSE;
			//				eStatoDosaggio := eST_COMPLETATO;
			//
			//			ELSIF TON_Stabilizzazione.Q THEN
			//				// 2. Controllo di errore: Timeout raggiunto
			//
			//				bStartTimer := FALSE; // Spegne il timer
			//				bErroreStabilizzazione := TRUE; // Segnala l'errore specifico
			//				eStatoDosaggio := eST_ERRORE;
			//
			//				// --- LOGICA DI AUTO-TARATURA ---
			//				// 1. Registra l'ultimo risultato e calcola l'errore
			//				fUltimoPesoDosato := fPesoAttualeBilancia;
			//				fUltimoErroreAssoluto := fUltimoPesoDosato - fPesoRichiesto; // Errore = (Finale - Richiesto)
			//
			//				// 2. Aggiorna il peso di anticipo chiusura (fPesoAnticipoChiusura)
			//				// Se l'ultimo dosaggio ha superato il setpoint (sovradosaggio):
			//				// L'errore è positivo, quindi dobbiamo aumentare l'anticipo (chiudere prima).
			//				// Nuova anticipazione = Vecchia anticipazione + (Errore * Fattore di correzione)
			//				fPesoAnticipoChiusura := fPesoAnticipoChiusura + (fUltimoErroreAssoluto * fFattoreCorrezione);
			//			END_IF

		eST_COMPLETATO: // Dosaggio terminato con successo
			bStartTimer := FALSE; // Timer disattivo
			bDosaggioCompletato := TRUE;
			bDosaggioInCorso := FALSE;
			fUscitaValvolaProporzionale := 0.0; // Valvola chiusa

			// --- LOGICA DI AUTO-TARATURA ---
			// 1. Registra l'ultimo risultato e calcola l'errore
			fUltimoPesoDosato := fPesoAttualeBilancia;
			fUltimoErroreAssoluto := fUltimoPesoDosato - fPesoRichiesto; // Errore = (Finale - Richiesto)

			// 2. Aggiorna il peso di anticipo chiusura (fPesoAnticipoChiusura)
			// Se l'ultimo dosaggio ha superato il setpoint (sovradosaggio):
			// L'errore è positivo, quindi dobbiamo aumentare l'anticipo (chiudere prima).
			// Nuova anticipazione = Vecchia anticipazione + (Errore * Fattore di correzione)
			fPesoAnticipoChiusura := fPesoAnticipoChiusura + (fUltimoErroreAssoluto * fFattoreCorrezione);

			// Limitare l'anticipo per evitare che diventi negativo o eccessivo (es. tra 1g e 100g)
			IF fPesoAnticipoChiusura < 1.0 THEN
				fPesoAnticipoChiusura := 1.0;
			END_IF

			// Ritorna in IDLE solo se il comando di avvio è disattivato
			IF NOT bAvviaDosaggio THEN
				eStatoDosaggio := eST_IDLE;
			END_IF

		eST_ERRORE: // Stato di errore (aggiungere logica di gestione errori più specifica)
			bStartTimer := FALSE; // Timer disattivo
			fUscitaValvolaProporzionale := 0.0;
			bDosaggioInCorso := FALSE;
			bStartTimerAttesa := FALSE;

			IF NOT bAvviaDosaggio THEN
				eStatoDosaggio := eST_IDLE;
			END_IF

	END_CASE

	fPesoAnticipoChiusura := fTempoRitardoPrecedente;

	// Calcolo e monitoraggio dell'errore (solo per info esterna/HMI)
	IF fPesoAttualeBilancia > 0.0 AND fPesoRichiesto > 0.0 THEN
		fErrorePercentuale := ABS((fPesoAttualeBilancia - fPesoRichiesto) / fPesoRichiesto) * 100.0;
	ELSE
		fErrorePercentuale := 0.0;
	END_IF

END_FUNCTION_BLOCK

FUNCTION_BLOCK FB_GestioneBilancia
	// 1. Determinazione del Range Raw (Mapping Raw Minimo)
	CASE eTipoSegnale OF
		eST_0_20mA:
			iRawMin := 0; // 0mA corrisponde al minimo raw (0)
			bErroreSegnale := FALSE; // Non c'è errore di "live zero"

		eST_4_20mA:
			// Calcolo il valore raw corrispondente a 4mA
			// (4mA / 20mA) * RawMax = 0.2 * RawMax
			iRawMin := REAL_TO_INT(iRawMax * 0.2) ;

			// Controllo errore segnale (Live Zero Check)
			IF iRawInput < iRawMin - 100 THEN // Sotto la soglia di 4mA (tolleranza 100 counts)
				bErroreSegnale := TRUE;
			ELSE
				bErroreSegnale := FALSE;
			END_IF
	END_CASE

	// 2. Calcolo del Fattore di Conversione e del Peso Lordo (fPesoLordoSenzaOffset)

	// Calcolo del range effettivo del segnale in Raw
	iRawRange := iRawMax - iRawMin;
	fRawAttualeNormalizzato := INT_TO_REAL(iRawInput) - INT_TO_REAL(iRawMin);

	// Se il range è valido
	IF iRawRange > 0 THEN
		// Fattore di conversione: Capacità / Range Raw
		fFattoreConversione := fCapacitaMaxG / INT_TO_REAL(iRawRange);

		// Peso Lordo = Raw Normalizzato * Fattore Conversione
		fPesoLordoSenzaOffset := fRawAttualeNormalizzato * fFattoreConversione;
	ELSE
		fPesoLordoSenzaOffset := 0.0;
	END_IF

	// 3. Gestione del Comando di Tara (Azzeramento)
	// La tara viene applicata al peso Lordo solo se il comando è attivo E non c'è errore di segnale
	IF bComandoTare AND NOT bErroreSegnale THEN
		fOffsetTara := fPesoLordoSenzaOffset;
	END_IF

	// 4. Calcolo del Peso Netto (Peso Lordo - Offset Tara)
	fPesoGrammi := fPesoLordoSenzaOffset - fOffsetTara;

	// Misure di sicurezza: Impedisci output troppo negativo
	IF fPesoGrammi < -15.0 THEN
		fPesoGrammi := 0.0;
	END_IF

END_FUNCTION_BLOCK
```

### Program Logical/Recipe (IEC)

#### Variables.var
```iecst
VAR
	MpRecipeXml_0 : MpRecipeXml;
	MpRecipeRegPar_0 : MpRecipeRegPar;
	UIConnect : MpRecipeUIConnectType;
	UISetup : MpRecipeUISetupType;
	MpRecipeUI_0 : MpRecipeUI;
END_VAR
```

#### Cyclic.ld
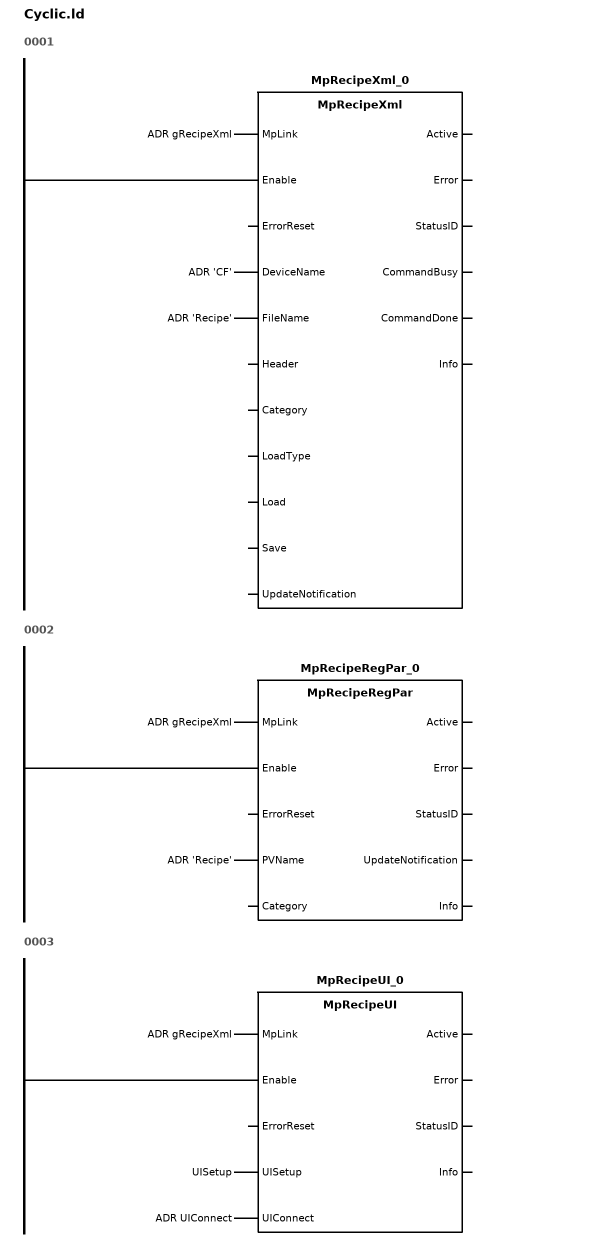
Ladder, written as Structured Text:
```iecst
PROGRAM _CYCLIC
(* Network 1 *)
MpRecipeXml_0(MpLink := ADR(gRecipeXml), Enable := TRUE, DeviceName := ADR('CF'), FileName := ADR('Recipe'));

(* Network 2 *)
MpRecipeRegPar_0(MpLink := ADR(gRecipeXml), Enable := TRUE, PVName := ADR('Recipe'));

(* Network 3 *)
MpRecipeUI_0(MpLink := ADR(gRecipeXml), Enable := TRUE, UISetup := UISetup, UIConnect := ADR(UIConnect));
END_PROGRAM
```

- Visualisation Logical/mappView (not shown)

### Program Logical/simu (IEC)

#### Variables.var
```iecst
VAR
	VelocitaValvola : REAL;
	peso : REAL;
END_VAR
```

#### Cyclic.st
```iecst
PROGRAM _CYCLIC
	(* Insert code here *)
	VelocitaValvola := (32767.0-6553.0)/700.0;

	IF (GlbIO.Ao.Valvola - GlbIO.Ai.Valvola) >= 500 THEN
		GlbIO.Ai.Valvola := GlbIO.Ai.Valvola + REAL_TO_INT(VelocitaValvola);
	ELSIF (GlbIO.Ao.Valvola - GlbIO.Ai.Valvola) < 500 THEN
		GlbIO.Ai.Valvola := GlbIO.Ai.Valvola - REAL_TO_INT(VelocitaValvola);
	END_IF

	IF GlbIO.Ai.Valvola > 6660 THEN
		//PesoBilancia_G := PesoBilancia_G + (50.0 * INT_TO_REAL(GlbIO.Ai.Valvola) / 32767.0);
		peso := peso + (5.0 * INT_TO_REAL(GlbIO.Ai.Valvola) / 32767.0);
	END_IF

	PesoBilancia_G := peso;

END_PROGRAM
```

Listed in the project but not available here: Logical/Program/Exit.st
